Staubli VAL3: init.pgx

public program init(num x_nDetNum (dimensions=1), string x_sTask (dimensions=1))
  local num l_i
  local bool l_bReport
  local num l_nLibNum
  local num l_nSocketIndex
  local string l_sLibName
begin
  //***** Customizable section
  //
  //***** end of customizable section
  // ************************
  // do not change anything beyond this line
  //
  //***************************
  //********* Strings *********
  //***************************
  sTASK=x_sTask+toString("",x_nDetNum)
  sDetNum="DET"+toString("",x_nDetNum)
  //
  //***************************
  //*****   Numerics     ******
  //***************************
  // Number of detected objects
  nNumOfPart=-1
  //
  // Resize buffers
  resize(nObjectID,1,nMaxNumOfObject)
  resize(nLatchedValue,1,nMaxNumOfObject)
  resize(trObjectPos,1,nMaxNumOfObject)
  resize(oTempQueue,1,nMaxNumOfObject)
  //
  // Initialize ID buffer
  for l_i=0 to size(nObjectID)-1
    nObjectID[l_i]=-1
  endFor
  //
  // Initialize Latched Encoder Value buffer
  for l_i=0 to size(nLatchedValue)-1
    nLatchedValue[l_i]=0
  endFor
  //
  // Initialize TRSF buffer
  for l_i=0 to size(trObjectPos)-1
    trObjectPos[l_i]={0,0,0,0,0,0}
  endFor
  //
  //***************************
  //*****   Booleans     ******
  //***************************
  // Detection library in calibration mode.
  //  Only used by the detection library "Socket".
  bCalibrating=false
  //
  //***************************
  //********* Sockets *********
  //***************************
  // Read the number of the library (ex. Cognex1 or Cognex2)
  call ut:getLibName(libPath(),l_sLibName)
  toNum(delete(l_sLibName,6,0),l_nLibNum,l_bReport)
  if !l_bReport
    l_nLibNum=1
  endIf
  l_nSocketIndex=l_nLibNum-1
  // Link socket
  sioLink(skVision,sck:skCognex[l_nSocketIndex])
  //
end
